// TIA Portal V19 export
DATA_BLOCK "instCallProjectSimulation"   // DB139
// stored: InstanceOfName CallProjectSimulation, InstanceOfType FB
"CallProjectSimulation"
   // VAR
   //    statNextStepBool : Bool;
   //    statCurrentStep : DInt;
   //    statInit : Bool;
   //    statStop : Bool;
   //    statReset : Bool;
   //    statNextStepBoolPre : Bool;
   //    ack : Bool;
   //    U2EM1setSingleStepMode : Bool;
   //    U2EM1nextStep : Bool;
   //    U2EM2setSingleStepMode : Bool;
   //    U2EM2nextStep : Bool;
   //    U2EM3setSingleStepMode : Bool;
   //    U2EM3nextStep : Bool;
   //    U2EM4setSingleStepMode : Bool;
   //    U2EM4nextStep : Bool;
   //    U2EM5setSingleStepMode : Bool;
   //    U2EM5nextStep : Bool;
   //    U2EM6setSingleStepMode : Bool;
   //    U2EM6nextStep : Bool;
   //    U2EM1Step : DInt;
   //    U2EM2Step : DInt;
   //    U2EM3Step : DInt;
   //    U2EM4Step : DInt;
   //    U2EM5Step : DInt;
   //    U2EM6Step : DInt;
   //    U2EM1cm1Vfd205 : "LEXCHANGETRAY_typeRollerVfdInterface";
   //    U2EM1cm2SingalTM : "LEXCHANGETRAY_typeRollerIoSignalInterface";
   //    U2EM2cm1Vfd206 : "LEXCHANGETRAY_typeRollerVfdInterface";
   //    U2EM2cm1Vfd { S7_SetPoint := 'True'} : "LEXCHANGETRAY_typeVfdInterface";
   //    U2EM2cm2TrayLiftingCylinder { S7_SetPoint := 'True'} : "LBC_Simple_typeTwoWayActuatorInterface";
   //    U2EM2cm3CellLiftingCylinder { S7_SetPoint := 'True'} : "LBC_Simple_typeTwoWayActuatorInterface";
   //    U2EM2cm4PositioningPinCylinder { S7_SetPoint := 'True'} : "LBC_Simple_typeTwoWayActuatorInterface";
   //    U2EM2cm5AxisControl { S7_SetPoint := 'True'} : "LBC_typeAxisSimpleControlNode_1";
   //    U2EM2cm6SignalTM { S7_SetPoint := 'True'} : "LEXCHANGETRAY_typeConstraintRollerIoSignalInterface";
   //    U2EM2cm7Pc { S7_SetPoint := 'True'} : "LEXCHANGETRAY_typePc_Interface";
   //    U2EM2cm8Scanner { S7_SetPoint := 'True'} : "LEXCHANGETRAY_typeSR1000Interface";
   //    U2EM3cm1SV112_Constraint1_Axis { S7_SetPoint := 'True'} : "LBC_typeAxisSimpleControlNode_1";
   //    U2EM3cm2SV113_Constraint2_Axis { S7_SetPoint := 'True'} : "LBC_typeAxisSimpleControlNode_1";
   //    U2EM3cm3SV115_Screw1_Axis : "LEXCHANGETRAY_typeAxisSimpleControlNode_2";
   //    U2EM3cm4SV116_Screw2_Axis : "LEXCHANGETRAY_typeAxisSimpleControlNode_2";
   //    U2EM3cm6SlideCylinder1 { S7_SetPoint := 'True'} : "LBC_Simple_typeTwoWayActuatorInterface";
   //    U2EM3cm7hookClawCylinder1 { S7_SetPoint := 'True'} : "LBC_Simple_typeTwoWayActuatorInterface";
   //    U2EM3cm8SlideCylinder2 { S7_SetPoint := 'True'} : "LBC_Simple_typeTwoWayActuatorInterface";
   //    U2EM3cm9hookClawCylinder2 { S7_SetPoint := 'True'} : "LBC_Simple_typeTwoWayActuatorInterface";
   //    U2EM3cm10SignalTM { S7_SetPoint := 'True'} : "LEXCHANGETRAY_typeConstraintWorkstationIoSignalInterface";
   //    U2EM3cm11PressureGaugeRs485 { S7_SetPoint := 'True'} : "typePressureGuageRs485Interface";
   //    statIndex { S7_SetPoint := 'True'} : Int;
   //    errors { S7_SetPoint := 'True'} : Array[0..9] of Int;
   //    timer1 : Array[0..23] of TON_TIME;
   // END_VAR
BEGIN
END_DATA_BLOCK
